// TIA Portal V19 export
FUNCTION "A04_HMI_CALL" : Void   // FC255, LAD
// stored: SetENOAutomatically false
BEGIN

REGION Network 1
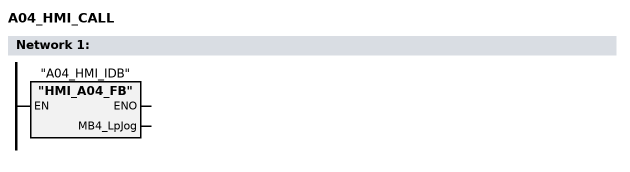
   RUNG wire#powerrail
      "A04_HMI_IDB"(MB4_LpJog =>)
   END_RUNG
   // the same network as SCL:
   "A04_HMI_IDB"();   // "HMI_A04_FB"
END_REGION
END_FUNCTION
